INTERFACE I_EventHandlerItem

METHOD PUBLIC Dispose
VAR_INPUT
END_VAR
END_METHOD

METHOD PUBLIC Emit
VAR_INPUT
	Event : I_Event;
END_VAR
END_METHOD

METHOD EqualTo : BOOL
VAR_INPUT
	Handler : I_EventHandler;
END_VAR
END_METHOD

PROPERTY PUBLIC Next : I_EventHandlerItem
GET
END_GET
SET
END_SET
END_PROPERTY

PROPERTY PUBLIC Previous : I_EventHandlerItem
GET
END_GET
SET
END_SET
END_PROPERTY

END_INTERFACE

(* stored: Version 1.1.0.1, ProductVersion 3.1.4024.12
   Itf I_EventHandlerItem: Id {037216c6-6832-0ae9-1b5c-d8b16d4eeb74}
   Method Dispose: Id {2e2e2368-d300-0481-0b4a-5718d3296ac6}
   Method Emit: Id {4330b441-0e47-0191-0c5e-1f386aed800a}
   Method EqualTo: Id {891a4d19-2c72-038b-23f8-e2e209915aee}
   Property Next: Id {627a2d51-95db-0623-07e1-f0509f61c220}
   Get Get: Id {953a37d0-697f-0bde-089d-3d6286ece612}
   Set Set: Id {a528daef-ab37-081d-2e73-788151168a4d}
   Property Previous: Id {00dccaee-c97f-0e4b-13c8-ca1ccdb30b61}
   Get Get: Id {dd25a8df-5486-0379-31bc-0f2356762499}
   Set Set: Id {2184d856-4c61-0e44-3085-c75967a1cbb6} *)
